// TIA Portal V15.1 export
// export: Created 2020-06-12T07:35:54.1630859Z, ExportSetting None, DisplayName Totally Integrated Automation Portal, DisplayVersion V15.1, DisplayName TIA Portal Openness, DisplayVersion V15.1, DisplayName STEP 7 Professional, DisplayVersion V15.1, DisplayName STEP 7 Safety, DisplayVersion V15.1, DisplayName WinCC Advanced, DisplayVersion V15.1
FUNCTION "RCW_main" : Void   // FC183, FBD
TITLE = RCW main
{ S7_Optimized_Access := 'TRUE' }
// stored: SetENOAutomatically False
   VAR_TEMP
      tStop : Bool;
      tStart : Bool;
      tStartFan : Bool;
      tStopFan : Bool;
   END_VAR
BEGIN

REGION Network 1: HMI request treat
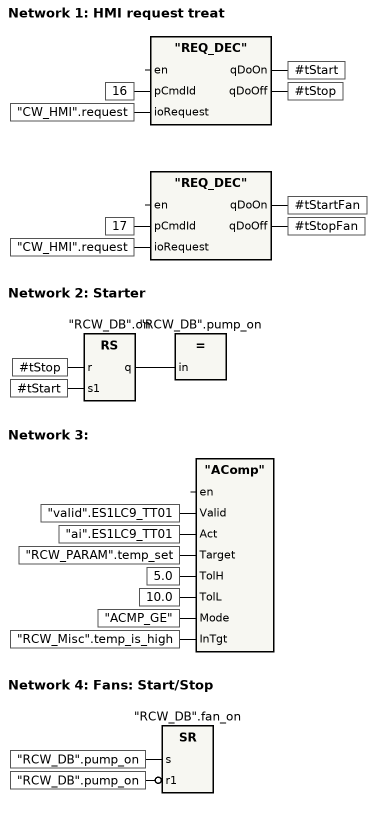
   "REQ_DEC"(pCmdId := 16, ioRequest := "CW_HMI".request, qDoOn => #tStart, qDoOff => #tStop);
   "REQ_DEC"(pCmdId := 17, ioRequest := "CW_HMI".request, qDoOn => #tStartFan, qDoOff => #tStopFan);
END_REGION

REGION Network 2: Starter
   IF #tStop THEN
       "RCW_DB".on := FALSE;   // RS flip-flop
   END_IF;
   IF #tStart THEN "RCW_DB".on := TRUE; END_IF;
   "RCW_DB".pump_on := "RCW_DB".on;
END_REGION

REGION Network 3
   "AComp"(Valid := "valid".ES1LC9_TT01,
           Act := "ai".ES1LC9_TT01,
           Target := "RCW_PARAM".temp_set,
           TolH := 5.0,
           TolL := 10.0,
           Mode := "ACMP_GE",
           InTgt := "RCW_Misc".temp_is_high);
END_REGION

REGION Network 4: Fans: Start/Stop
   IF "RCW_DB".pump_on THEN
       "RCW_DB".fan_on := TRUE;   // SR flip-flop
   END_IF;
   IF NOT "RCW_DB".pump_on THEN "RCW_DB".fan_on := FALSE; END_IF;
END_REGION

REGION Network 5: HMI: STATUS
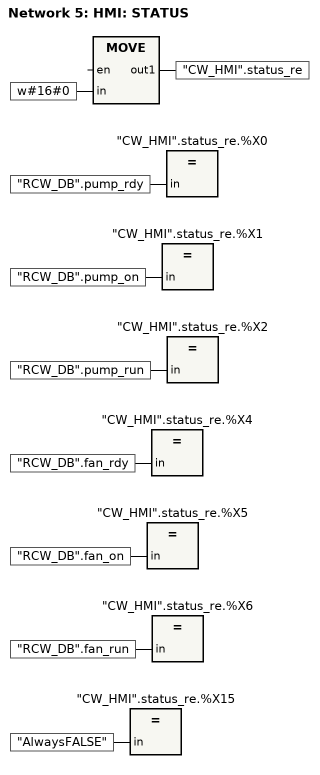
   "CW_HMI".status_re := w#16#0;
   "CW_HMI".status_re.%X0 := "RCW_DB".pump_rdy;
   "CW_HMI".status_re.%X1 := "RCW_DB".pump_on;
   "CW_HMI".status_re.%X2 := "RCW_DB".pump_run;
   "CW_HMI".status_re.%X4 := "RCW_DB".fan_rdy;
   "CW_HMI".status_re.%X5 := "RCW_DB".fan_on;
   "CW_HMI".status_re.%X6 := "RCW_DB".fan_run;
   "CW_HMI".status_re.%X15 := "AlwaysFALSE";
END_REGION
END_FUNCTION
